PROGRAM MAIN
VAR
	motor	 			: ACMotor;
	motorChangeTimer 	: TON;
	
	startButton			: ButtonNC;
	signalTower			: SignalTower;
END_VAR

MotionLogic();
SignalTowerLogic();

METHOD MotionLogic
IF startButton.IsPressed THEN
	motorChangeTimer(
		IN := NOT motorChangeTimer.Q,
		PT := T#10S);
	
	IF motorChangeTimer.Q AND_THEN motor.IsMoving THEN
		motor.Stop();
	ELSIF motorChangeTimer.Q THEN
		motor.Start();
	END_IF
ELSE
	motorChangeTimer(IN := FALSE);
	motor.Stop();
END_IF
END_METHOD

METHOD SignalTowerLogic
VAR_INPUT
END_VAR
IF startButton.IsPressed THEN
	signalTower.SetStateOP();
ELSE
	signalTower.SetStateSTOP();
END_IF
END_METHOD

END_PROGRAM

(* stored: Version 1.1.0.1, ProductVersion 3.1.4024.12
   POU MAIN: Id {c893af56-82c6-43a2-a7ff-57a3ef97d3b2}, SpecialFunc None
   Method MotionLogic: Id {2193b283-ee17-414b-be29-95a0081b03c1}
   Method SignalTowerLogic: Id {42ff7a04-4492-40ce-b4e2-ee240cf33ede} *)
